INTERFACE I_Area2Robot

//{attribute 'monitoring' := 'variable'}
{attribute 'monitoring' := 'call'}
PROPERTY Busy : BOOL
GET
END_GET
END_PROPERTY

METHOD clearCommand : BOOL
VAR_INPUT
END_VAR
END_METHOD

//{attribute 'monitoring' := 'variable'}
{attribute 'monitoring' := 'call'}
PROPERTY Done : BOOL
GET
END_GET
END_PROPERTY

{attribute 'monitoring' := 'call'}
PROPERTY Ready : BOOL
GET
END_GET
END_PROPERTY

METHOD release : BOOL
VAR_INPUT
	sectionReservation : SectionEnum;
END_VAR
END_METHOD

METHOD reserve : BOOL
VAR_INPUT
	reserveRequest : SectionEnum;
END_VAR
(*
this method exists because chipboard and wood bunk operations use the same robot
both sections need to check if the robot is open to commands before use
*)
END_METHOD

{attribute 'monitoring' := 'call'}
PROPERTY Reserved : BOOL
GET
END_GET
END_PROPERTY

METHOD reset : BOOL
END_METHOD

METHOD stop : BOOL
VAR_INPUT
END_VAR
END_METHOD

END_INTERFACE

(* stored: Version 1.1.0.1, ProductVersion 3.1.4024.11
   Itf I_Area2Robot: Id {81769b72-e253-4c65-bc45-fd00894d820b}
   Folder Properties: Id {48ccb73b-0acd-4bff-b234-48ccbf283e2d}
   Property Busy: Id {4c468d72-c4ac-4a81-a1cb-e703e9390365}
   Get Get: Id {3a934247-7cc8-490d-9719-9702872fe1ac}
   Method clearCommand: Id {383c1c5a-b200-4238-8619-fb67560d9a76}
   Property Done: Id {129a1422-6b89-43b1-a482-13337fd43d30}
   Get Get: Id {647a1ab6-cf6c-45fb-8853-b2ad79ffcea5}
   Property Ready: Id {338c913a-eef0-4be2-b7c0-4bc891ba978d}
   Get Get: Id {8806150f-43fd-4064-8b9b-f2e383fe3af6}
   Method release: Id {f4f4d439-0be9-4890-bec6-ec93c43ed77c}
   Method reserve: Id {06446207-c0c4-403e-a233-848eb7b14014}
   Property Reserved: Id {c231ade8-8ccf-4d42-bdf8-b42b42aa80f0}
   Get Get: Id {38f84467-ee49-41c3-8b98-c46381301cd8}
   Method reset: Id {2d52e7f4-06eb-4793-a855-2ba59843e286}
   Method stop: Id {5bdcbd02-0470-4035-ac1a-b4a6b831f0d8} *)
